(* PLC project Tc2_IoFunctions.F_CreateDpv1ReadReqPkg Demo, tc3-libraries-kb TwinCAT 3.1 *)
(* stored: creationDateTime 2026-05-21T00:00:00, modificationDateTime 2026-05-21T00:00:00 *)

PROGRAM P_Demo_F_CreateDpv1ReadReqPkg
  VAR
    aDpv1ReqBuffer : ARRAY[1..240] OF BYTE;  (* DPV1 读请求帧缓冲 240 字节 *)
    arrDpv1ReqParams : ARRAY[1..39] OF ST_Dpv1ParamAddrEx;  (* 参数清单 *)
    iNumParamsToRead : USINT := 3;  (* 要读的参数数 *)
    iDriveObjectId : USINT := 2;  (* 1=CU 2=drive A 3=drive B *)
    bBuildReqPkg : BOOL := FALSE;  (* 触发：构造请求帧 *)
    nReqPkgLen : USINT;  (* 生成的帧长度（字节） *)
  END_VAR

// =============================================================================
// 场景：SINAMICS S120 上电诊断：构造一个 DPV1 读请求帧读取 3 个驱动器参数。
// 价值：把 DPV1 帧手撸协议替换为函数调用。
// 验证：登录后填好 arrDpv1ReqParams[1..3]（每条含 parameter number + sub-index + length），写 bBuildReqPkg := TRUE → 一个 PLC 周期后 nReqPkgLen 显示生成的帧长度（> 0 表示成功）。
// 验证步骤：
//   1. 右键 PLC 项目 → Import PLCopenXML → 选本文件
//   2. 引用 Tc2_IoFunctions（References → Add library）
//   3. 编译 → 登录 → 运行；按上方『验证』行的指示在线写值观察
// =============================================================================

// 单次调用：构造帧，立即返回长度
IF bBuildReqPkg THEN
    nReqPkgLen := F_CreateDpv1ReadReqPkg(
        pDpv1ReqData    := ADR(aDpv1ReqBuffer),
        iNumOfParams    := iNumParamsToRead,
        iDriveId        := iDriveObjectId,
        stDpv1Parameter := arrDpv1ReqParams
    );
    bBuildReqPkg := FALSE;
END_IF;
END_PROGRAM
